FUNCTION_BLOCK AnalogInputBase (* Composite Function Block Type *)
  (* Standard: 61499-2 *)
  (* Version 1.0.1, 1/16/2024, ApplicationLibDevTeam, Schneider Electric, First Version *)
  PACKAGE SE.Nereda;
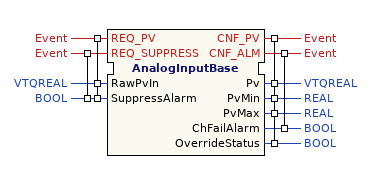
  EVENT_INPUT
    REQ_PV WITH RawPvIn, SuppressAlarm; (* Request input value *)
    REQ_SUPPRESS WITH SuppressAlarm; (* Request to suppress the channel failure alarm *)
  END_EVENT
  EVENT_OUTPUT
    CNF_PV WITH Pv, PvMin, PvMax, OverrideStatus; (* Execution confirmation of Pv *)
    CNF_ALM WITH ChFailAlarm; (* Execution confirmation of alarm *)
  END_EVENT
  VAR_INPUT
    RawPvIn : VTQREAL; (* Unscaled analog signal *)
    SuppressAlarm : BOOL; (* 1 = Suppress channel failure in HMI *)
  END_VAR
  VAR_OUTPUT
    Pv : VTQREAL; (* Scaled process signal *)
    PvMin : REAL; (* Minimum pv measurement range (in engineering units) *)
    PvMax : REAL; (* Maximun pv measurement range (in engineering units) *)
    ChFailAlarm : BOOL; (* 1 = Alarm condition is true with considering the suppress status *)
    OverrideStatus : BOOL; (* 1 = Signal is forced from HwCat based on quality code *)
  END_VAR
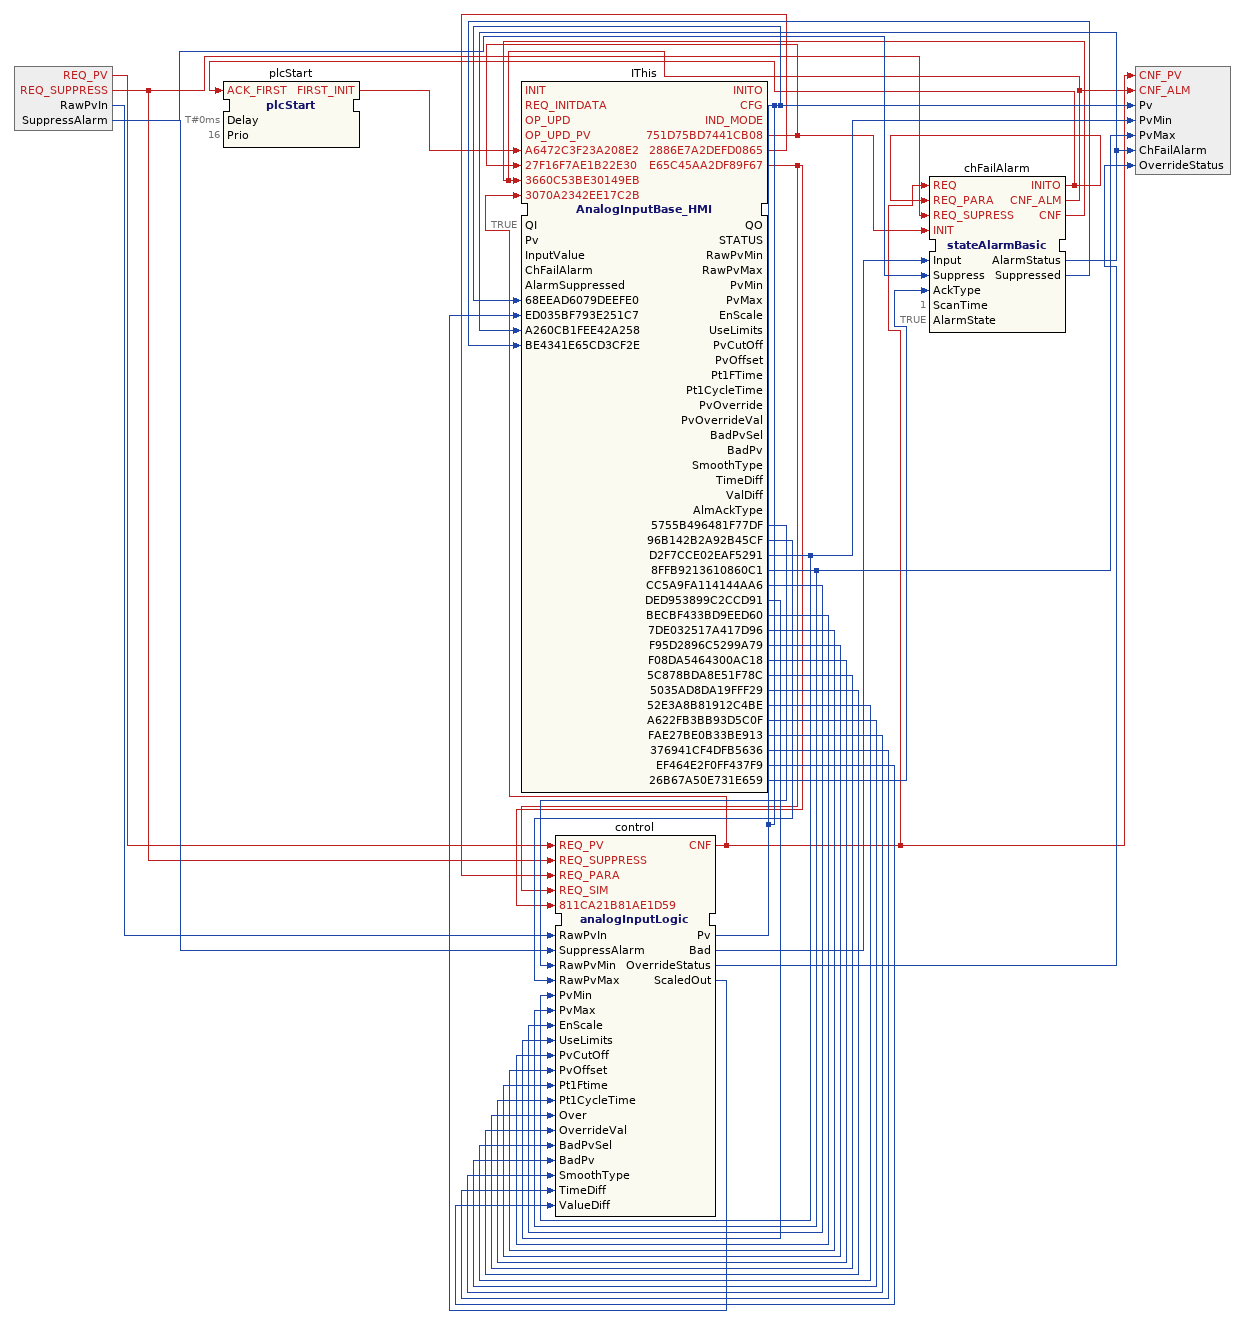
  (* Initialization *)
  (* HMI *)
  (* Analog Input Core *)
  (* Alarm management *)
  FBS
    plcStart : plcStart(Delay := T#0ms, Prio := 16);
    IThis : AnalogInputBase_HMI(QI := TRUE); {SET_ATTRIBUTE(Configuration.Component.HideUnusedPorts, )}
    control : analogInputLogic;
    chFailAlarm : stateAlarmBasic(ScanTime := 1, AlarmState := TRUE); {SET_ATTRIBUTE(HMI.AlarmText, $key:SE.App2CommonProcess.TxtSignalFail)}
  END_FBS
  EVENT_CONNECTIONS
    REQ_PV TO control.REQ_PV;
    control.CNF TO chFailAlarm.REQ;
    chFailAlarm.INITO TO plcStart.ACK_FIRST;
    REQ_SUPPRESS TO control.REQ_SUPPRESS;
    chFailAlarm.INITO TO chFailAlarm.REQ_PARA;
    REQ_SUPPRESS TO chFailAlarm.REQ_SUPRESS;
    control.CNF TO CNF_PV;
    chFailAlarm.CNF_ALM TO CNF_ALM;
    plcStart.FIRST_INIT TO IThis.A6472C3F23A208E2;
    IThis.751D75BD7441CB08 TO IThis.27F16F7AE1B22E30;
    chFailAlarm.CNF_ALM TO IThis.3660C53BE30149EB;
    chFailAlarm.CNF TO IThis.3660C53BE30149EB;
    control.CNF TO IThis.3070A2342EE17C2B;
    IThis.751D75BD7441CB08 TO chFailAlarm.INIT;
    IThis.2886E7A2DEFD0865 TO control.REQ_PARA;
    IThis.E65C45AA2DF89F67 TO control.REQ_SIM;
    IThis.E65C45AA2DF89F67 TO control.811CA21B81AE1D59;
  END_CONNECTIONS
  DATA_CONNECTIONS
    control.Pv TO Pv;
    RawPvIn TO control.RawPvIn;
    control.Bad TO chFailAlarm.Input;
    SuppressAlarm TO chFailAlarm.Suppress;
    SuppressAlarm TO control.SuppressAlarm;
    chFailAlarm.AlarmStatus TO ChFailAlarm;
    control.OverrideStatus TO OverrideStatus;
    control.Pv TO IThis.68EEAD6079DEEFE0;
    control.ScaledOut TO IThis.ED035BF793E251C7;
    chFailAlarm.AlarmStatus TO IThis.A260CB1FEE42A258;
    chFailAlarm.Suppressed TO IThis.BE4341E65CD3CF2E;
    IThis.5755B496481F77DF TO control.RawPvMin;
    IThis.96B142B2A92B45CF TO control.RawPvMax;
    IThis.D2F7CCE02EAF5291 TO PvMin;
    IThis.D2F7CCE02EAF5291 TO control.PvMin;
    IThis.8FFB9213610860C1 TO PvMax;
    IThis.8FFB9213610860C1 TO control.PvMax;
    IThis.CC5A9FA114144AA6 TO control.EnScale;
    IThis.DED953899C2CCD91 TO control.UseLimits;
    IThis.BECBF433BD9EED60 TO control.PvCutOff;
    IThis.7DE032517A417D96 TO control.PvOffset;
    IThis.F95D2896C5299A79 TO control.Pt1Ftime;
    IThis.F08DA5464300AC18 TO control.Pt1CycleTime;
    IThis.5C878BDA8E51F78C TO control.Over;
    IThis.5035AD8DA19FFF29 TO control.OverrideVal;
    IThis.52E3A8B81912C4BE TO control.BadPvSel;
    IThis.A622FB3BB93D5C0F TO control.BadPv;
    IThis.FAE27BE0B33BE913 TO control.SmoothType;
    IThis.376941CF4DFB5636 TO control.TimeDiff;
    IThis.EF464E2F0FF437F9 TO control.ValueDiff;
    IThis.26B67A50E731E659 TO chFailAlarm.AckType;
  END_CONNECTIONS
END_FUNCTION_BLOCK
